// SIMATIC STEP 7 (V5.x) project TF_TACHO_PROJECT
// CPU: CPU 315-2 DP
// station: Hardware
// station: SIMATIC 300
// station: P_ADR_BUS
// station: _S7H_BUSSYSTEM_CT
// program: S7 Program(1)

SYMBOL_TABLE
"DB_Entradas_Proceso"	DB 1	DB 1
"DB_Entradas_HMI"	DB 2	DB 2
"DB_Salidas_Proceso"	DB 3	DB 3
"DB_Salidas_HMI"	DB 4	DB 4
"DB_Flags_Fallas"	DB 5	DB 5
"DB_Aux"	DB 6	DB 6	// DB de variables auxiliares
"DB_Grafo_Marcha"	DB 7	FB 1
"DB_Grafo_ON_OFF"	DB 8	FB 2
"DB_Grafo_PID"	DB 9	FB 3
"DB_CTRL_GRAFOS"	DB 10	DB 10	// DB Global de estados y transiciones de grafos
"DB_PID"	DB 11	FB 41
"FB_Grafo_Marcha"	FB 1	FB 1
"FB_Grafo_ON_OFF"	FB 2	FB 2
"FB_Grafo_PID"	FB 3	FB 3
"CONT_C"	FB 41	FB 41	// Continuous Control
"FC_Init_constantes"	FC 1	FC 1
"FC_Manejo_Entradas_Proc"	FC 2	FC 2
"FC_Manejo_Entradas_HMI"	FC 3	FC 3
"FC_Modos_Operacion"	FC 4	FC 4
"FC_Calculo_Var_Aux"	FC 5	FC 5	// Funcion que calcula variables aux.
"FC_Adm_Fallas"	FC 6	FC 6	// Funcion que verifica fallas del sistema
"FC_Recuperacion_Fallas"	FC 7	FC 7	// Recuperacion automatica de fallas
"FC_Ctrl_ON_OFF"	FC 8	FC 8
"FC_Ctrl_PID"	FC 9	FC 9
"FC_Ctrl_Marcha"	FC 10	FC 10
"FC_Ejecucion_PID"	FC 11	FC 11
"G7_STD_3"	FC 72	FC 72
"SCALE"	FC 105	FC 105	// Scaling Values
"UNSCALE"	FC 106	FC 106	// Unscaling Values
"FALLA_BMB"	I 1.0	BOOL	// Señal (simulada) de falla de bomba
"NIV_SENS"	IW 0	INT	// Nivel sensado del liquido en el tacho (Cuentas)
"FALSE"	M 0.0	BOOL
"TRUE"	M 0.1	BOOL
"ALTURA_TACHO"	MD 1	REAL	// Altura del tacho (cm)
"NIVEL_ALTO"	MD 3	REAL	// Nivel maximo de agua en el tacho
"NIVEL_BAJO"	MD 5	REAL	// Minimo nivel de agua en el tacho
"Programa Principal"	OB 1	OB 1
"CYC_INT5"	OB 35	OB 35	// Cyclic Interrupt 5
"SALIDA_HL"	Q 4.0	BOOL	// Indicacion de nivel alto (HL)
"SALIDA_LL"	Q 4.1	BOOL	// Indicación de nivel bajo (LL)
"LUZ_MODO_OPER"	Q 4.2	BOOL	// Indicacion del modo de operacion (MANUAL-ON/OFF-PID)
"BMB_CARGA"	QW 0	WORD	// Señal de actuación sobre la bomba de carga del sistema. Rango entre 0 y 5 V.
"BMB_PERT"	QW 2	WORD	// Señal de actuación sobre la bomba de perturbación (vaciado) del sistema.
"TIME_TCK"	SFC 64	SFC 64	// Read the System Time
"VAT_SIM"	VAT 1	
END_SYMBOL_TABLE

FUNCTION_BLOCK "FB_Grafo_Marcha"	// FB 1
TITLE = S7GRAPH V4 FB
//Block comment
VERSION : 0.1
VAR_INPUT
  OFF_SQ : BOOL ;
  INIT_SQ : BOOL ;
  ACK_EF : BOOL ;
  S_PREV : BOOL ;
  S_NEXT : BOOL ;
  SW_AUTO : BOOL ;
  SW_TAP : BOOL ;
  SW_MAN : BOOL ;
  S_SEL : INT ;
  S_ON : BOOL ;
  S_OFF : BOOL ;
  T_PUSH : BOOL ;
END_VAR
VAR_OUTPUT
  S_NO : INT ;
  S_MORE : BOOL ;
  S_ACTIVE : BOOL ;
  ERR_FLT : BOOL ;
  AUTO_ON : BOOL ;
  TAP_ON : BOOL ;
  MAN_ON : BOOL ;
END_VAR
VAR
  G7T : ARRAY  [0 .. 3 ] OF STRUCT
   TV : BOOL ;
   TT : BOOL ;
   TS : BOOL ;
   CF_IV : BOOL ;
   TNO : INT ;
   CRIT : DWORD ;
   CRIT_OLD : DWORD ;
   CRIT_FLT : DWORD ;
  END_STRUCT ;
  G7S : ARRAY  [0 .. 3 ] OF STRUCT
   S1 : BOOL ;
   L1 : BOOL ;
   V1 : BOOL ;
   R1 : BOOL ;
   A1 : BOOL ;
   S0 : BOOL ;
   L0 : BOOL ;
   V0 : BOOL ;
   X : BOOL ;
   LA : BOOL ;
   VA : BOOL ;
   RA : BOOL ;
   AA : BOOL ;
   SS : BOOL ;
   LS : BOOL ;
   VS : BOOL ;
   SNO : INT ;
   T : TIME ;
   U : TIME ;
   CRIT_LOC : DWORD ;
   CRIT_LOC_ERR : DWORD ;
   CRIT_SUP : DWORD ;
   SM : BOOL ;
   LP : BOOL ;
   LN : BOOL ;
   VP : BOOL ;
   VN : BOOL ;
   H_IL_ERR : BYTE ;
   H_SV_FLT : BYTE ;
   RESERVED : DWORD ;
  END_STRUCT ;
  TVX : ARRAY  [0 .. 2 ] OF BYTE  := B#16#1;
  TTX : ARRAY  [0 .. 2 ] OF BYTE  := B#16#1;
  TSX : ARRAY  [0 .. 2 ] OF BYTE  := B#16#1;
  S00X : ARRAY  [0 .. 2 ] OF BYTE  := B#16#1;
  SOFFX : ARRAY  [0 .. 2 ] OF BYTE  := B#16#1;
  SONX : ARRAY  [0 .. 2 ] OF BYTE  := B#16#1;
  SAX : ARRAY  [0 .. 2 ] OF BYTE  := B#16#1;
  SERRX : ARRAY  [0 .. 4 ] OF BYTE  := B#16#1;
  SMX : ARRAY  [0 .. 4 ] OF BYTE  := B#16#1;
  S0X : ARRAY  [0 .. 4 ] OF BYTE  := B#16#1;
  S1X : ARRAY  [0 .. 4 ] OF BYTE  := B#16#1;
  S_DISPLAY : INT ;
  S_SEL_OLD : INT ;
  S_DISPIDX : BYTE ;
  T_DISPIDX : BYTE ;
  MOPEDGE : STRUCT
   AUTO : BOOL ;
   MAN : BOOL ;
   TAP : BOOL ;
   TOP : BOOL ;
   RES1 : BOOL ;
   RES2 : BOOL ;
   RES3 : BOOL ;
   RES4 : BOOL ;
   LOCK : BOOL ;
   SUP : BOOL ;
   ACKREQ : BOOL ;
   SSKIP : BOOL ;
   OFF : BOOL ;
   INIT : BOOL ;
   HALT : BOOL ;
   TMS_HALT : BOOL ;
   OPS_ZERO : BOOL ;
   SACT_DISP : BOOL ;
   SEF_DISP : BOOL ;
   SALL_DISP : BOOL ;
   S_PREV : BOOL ;
   S_NEXT : BOOL ;
   S_SELOK : BOOL ;
   S_ON : BOOL ;
   S_OFF : BOOL ;
   T_PUSH : BOOL ;
   REG : BOOL ;
   ACK : BOOL ;
   IL_PERM : BOOL ;
   T_PERM : BOOL ;
   ILP_MAN : BOOL ;
  END_STRUCT ;
  MOP : STRUCT
   AUTO : BOOL  := TRUE;
   MAN : BOOL ;
   TAP : BOOL ;
   TOP : BOOL ;
   RES1 : BOOL ;
   RES2 : BOOL ;
   RES3 : BOOL ;
   RES4 : BOOL ;
   LOCK : BOOL  := TRUE;
   SUP : BOOL  := TRUE;
   ACKREQ : BOOL  := TRUE;
   SSKIP : BOOL ;
   OFF : BOOL ;
   INIT : BOOL  := TRUE;
   HALT : BOOL ;
   TMS_HALT : BOOL ;
   OPS_ZERO : BOOL ;
   SACT_DISP : BOOL  := TRUE;
   SEF_DISP : BOOL ;
   SALL_DISP : BOOL ;
   S_PREV : BOOL ;
   S_NEXT : BOOL ;
   S_SELOK : BOOL ;
   S_ON : BOOL ;
   S_OFF : BOOL ;
   T_PUSH : BOOL ;
   REG : BOOL ;
   ACK : BOOL ;
   IL_PERM : BOOL ;
   T_PERM : BOOL ;
   ILP_MAN : BOOL ;
  END_STRUCT ;
  TICKS : STRUCT
   DELTA : TIME ;
   OLD : TIME ;
   NEW : TIME ;
  END_STRUCT ;
  SQ_FLAGS : STRUCT
   ERR_FLT : BOOL ;
   ERROR : BOOL ;
   FAULT : BOOL ;
   RT_FAIL : BOOL ;
   NO_SNO : BOOL ;
   NF_OFL : BOOL ;
   SA_OFL : BOOL ;
   TV_OFL : BOOL ;
   MSG_OFL : BOOL ;
   NO_SWI : BOOL ;
   CYC_OP : BOOL ;
   AS_MSG : BOOL ;
   AS_SEND : BOOL ;
   SQ_BUSY : BOOL ;
   SA_BUSY : BOOL ;
   AS_SIG : BOOL ;
  END_STRUCT ;
  S_PTR : DWORD  := DW#16#250;
  S_PTR2 : DWORD ;
  S_PTR3 : DWORD  := DW#16#7C0;
  S_PTR4 : DWORD  := DW#16#790;
  T_PTR : DWORD  := DW#16#760;
  C_AR2 : DWORD ;
  M_FBDB : DWORD  := DW#16#10000;
  M_SNO : WORD ;
  M_EVID : WORD ;
  M_EVIL : DWORD ;
  M_EVSV : DWORD ;
  M_EV : DWORD  := DW#16#6D0;
  CRIT : ARRAY  [0 .. 31 ] OF BOOL ;
  S_START : BYTE ;
  S_IDX : BYTE ;
  S_INT : INT  := 72;
  S_TMP : BYTE ;
  T_START : BYTE ;
  T_IDX : BYTE ;
  T_TMP : BYTE ;
  T_TMP2 : BYTE ;
  TV_POT : BYTE  := B#16#6;
  RETURN1 : BYTE ;
  RETURN2 : BYTE ;
  SINI : ARRAY  [0 .. 2 ] OF BYTE  := B#16#2, B#16#1;
  LSTT : ARRAY  [0 .. 3 ] OF BYTE  := B#16#0, B#16#0, B#16#0, B#16#2;
  ATAJ : ARRAY  [0 .. 3 ] OF BYTE  := B#16#0, B#16#1, B#16#2, B#16#3;
  ATAB : ARRAY  [0 .. 3 ] OF BYTE  := B#16#0, B#16#1, B#16#2, B#16#3;
  PSTT : ARRAY  [0 .. 3 ] OF BYTE  := B#16#0, B#16#1, B#16#2, B#16#3;
  NSTT : ARRAY  [0 .. 3 ] OF BYTE  := B#16#1, B#16#2, B#16#3, B#16#2;
  ASSJ : ARRAY  [0 .. 3 ] OF BYTE  := B#16#0, B#16#1, B#16#2, B#16#3;
  ASSB : ARRAY  [0 .. 3 ] OF BYTE  := B#16#0, B#16#1, B#16#2, B#16#3;
  PTTS : ARRAY  [0 .. 3 ] OF BYTE  := B#16#0, B#16#0, B#16#1, B#16#2;
  NTTS : ARRAY  [0 .. 3 ] OF BYTE  := B#16#0, B#16#1, B#16#2, B#16#3;
  PRE_CNT : WORD ;
  POST_CNT : WORD ;
  ADR_COND : WORD ;
  MAX_TVAL : BYTE  := B#16#1;
  MAX_SACT : BYTE  := B#16#1;
  MAX_CRIT : BYTE  := B#16#4;
  T_CNT : BYTE  := B#16#3;
  SUP_CNT : BYTE ;
  LOCK_CNT : BYTE ;
  S_CNT : BYTE  := B#16#3;
  SQ_CNT : BYTE  := B#16#1;
  PRS_INPAR : DWORD  := DW#16#E000F6C8;
  PRS_OUTPAR : DWORD  := DW#16#E000800D;
  GC_FLAGS : STRUCT
   T_MACH : WORD  := W#16#EB;
   COND_ED : WORD  := W#16#E3;
   W_LEVEL : WORD  := W#16#D5;
   AS_MSG : WORD ;
   FB_IF : WORD  := W#16#FC;
   SSB : WORD  := W#16#105;
   CRIT_AVAIL : BOOL ;
   SSKIP_AVAIL : BOOL  := TRUE;
   SSKIP_ON : BOOL ;
   ACK_REQ : BOOL  := TRUE;
   SYNC_AVAIL : BOOL ;
   ILP_MAN : BOOL ;
  END_STRUCT ;
  G7_FBMARK : BYTE  := B#16#25;
  G7_RELEASE : BYTE  := B#16#2A;
  G7_ID2 : BYTE  := B#16#37;
  G7_ID1 : BYTE  := B#16#47;
END_VAR
BEGIN
// body was compiled from an S7-GRAPH chart; compiled code not shown
END_FUNCTION_BLOCK

FUNCTION_BLOCK "FB_Grafo_ON_OFF"	// FB 2
TITLE = S7GRAPH V4 FB
//Block comment
VERSION : 0.1
VAR_INPUT
  OFF_SQ : BOOL ;
  INIT_SQ : BOOL ;
  ACK_EF : BOOL ;
  S_PREV : BOOL ;
  S_NEXT : BOOL ;
  SW_AUTO : BOOL ;
  SW_TAP : BOOL ;
  SW_MAN : BOOL ;
  S_SEL : INT ;
  S_ON : BOOL ;
  S_OFF : BOOL ;
  T_PUSH : BOOL ;
END_VAR
VAR_OUTPUT
  S_NO : INT ;
  S_MORE : BOOL ;
  S_ACTIVE : BOOL ;
  ERR_FLT : BOOL ;
  AUTO_ON : BOOL ;
  TAP_ON : BOOL ;
  MAN_ON : BOOL ;
END_VAR
VAR
  G7T : ARRAY  [0 .. 3 ] OF STRUCT
   TV : BOOL ;
   TT : BOOL ;
   TS : BOOL ;
   CF_IV : BOOL ;
   TNO : INT ;
   CRIT : DWORD ;
   CRIT_OLD : DWORD ;
   CRIT_FLT : DWORD ;
  END_STRUCT ;
  G7S : ARRAY  [0 .. 3 ] OF STRUCT
   S1 : BOOL ;
   L1 : BOOL ;
   V1 : BOOL ;
   R1 : BOOL ;
   A1 : BOOL ;
   S0 : BOOL ;
   L0 : BOOL ;
   V0 : BOOL ;
   X : BOOL ;
   LA : BOOL ;
   VA : BOOL ;
   RA : BOOL ;
   AA : BOOL ;
   SS : BOOL ;
   LS : BOOL ;
   VS : BOOL ;
   SNO : INT ;
   T : TIME ;
   U : TIME ;
   CRIT_LOC : DWORD ;
   CRIT_LOC_ERR : DWORD ;
   CRIT_SUP : DWORD ;
   SM : BOOL ;
   LP : BOOL ;
   LN : BOOL ;
   VP : BOOL ;
   VN : BOOL ;
   H_IL_ERR : BYTE ;
   H_SV_FLT : BYTE ;
   RESERVED : DWORD ;
  END_STRUCT ;
  TVX : ARRAY  [0 .. 2 ] OF BYTE  := B#16#1;
  TTX : ARRAY  [0 .. 2 ] OF BYTE  := B#16#1;
  TSX : ARRAY  [0 .. 2 ] OF BYTE  := B#16#1;
  S00X : ARRAY  [0 .. 2 ] OF BYTE  := B#16#1;
  SOFFX : ARRAY  [0 .. 2 ] OF BYTE  := B#16#1;
  SONX : ARRAY  [0 .. 2 ] OF BYTE  := B#16#1;
  SAX : ARRAY  [0 .. 2 ] OF BYTE  := B#16#1;
  SERRX : ARRAY  [0 .. 4 ] OF BYTE  := B#16#1;
  SMX : ARRAY  [0 .. 4 ] OF BYTE  := B#16#1;
  S0X : ARRAY  [0 .. 4 ] OF BYTE  := B#16#1;
  S1X : ARRAY  [0 .. 4 ] OF BYTE  := B#16#1;
  S_DISPLAY : INT ;
  S_SEL_OLD : INT ;
  S_DISPIDX : BYTE ;
  T_DISPIDX : BYTE ;
  MOPEDGE : STRUCT
   AUTO : BOOL ;
   MAN : BOOL ;
   TAP : BOOL ;
   TOP : BOOL ;
   RES1 : BOOL ;
   RES2 : BOOL ;
   RES3 : BOOL ;
   RES4 : BOOL ;
   LOCK : BOOL ;
   SUP : BOOL ;
   ACKREQ : BOOL ;
   SSKIP : BOOL ;
   OFF : BOOL ;
   INIT : BOOL ;
   HALT : BOOL ;
   TMS_HALT : BOOL ;
   OPS_ZERO : BOOL ;
   SACT_DISP : BOOL ;
   SEF_DISP : BOOL ;
   SALL_DISP : BOOL ;
   S_PREV : BOOL ;
   S_NEXT : BOOL ;
   S_SELOK : BOOL ;
   S_ON : BOOL ;
   S_OFF : BOOL ;
   T_PUSH : BOOL ;
   REG : BOOL ;
   ACK : BOOL ;
   IL_PERM : BOOL ;
   T_PERM : BOOL ;
   ILP_MAN : BOOL ;
  END_STRUCT ;
  MOP : STRUCT
   AUTO : BOOL  := TRUE;
   MAN : BOOL ;
   TAP : BOOL ;
   TOP : BOOL ;
   RES1 : BOOL ;
   RES2 : BOOL ;
   RES3 : BOOL ;
   RES4 : BOOL ;
   LOCK : BOOL  := TRUE;
   SUP : BOOL  := TRUE;
   ACKREQ : BOOL  := TRUE;
   SSKIP : BOOL ;
   OFF : BOOL ;
   INIT : BOOL  := TRUE;
   HALT : BOOL ;
   TMS_HALT : BOOL ;
   OPS_ZERO : BOOL ;
   SACT_DISP : BOOL  := TRUE;
   SEF_DISP : BOOL ;
   SALL_DISP : BOOL ;
   S_PREV : BOOL ;
   S_NEXT : BOOL ;
   S_SELOK : BOOL ;
   S_ON : BOOL ;
   S_OFF : BOOL ;
   T_PUSH : BOOL ;
   REG : BOOL ;
   ACK : BOOL ;
   IL_PERM : BOOL ;
   T_PERM : BOOL ;
   ILP_MAN : BOOL ;
  END_STRUCT ;
  TICKS : STRUCT
   DELTA : TIME ;
   OLD : TIME ;
   NEW : TIME ;
  END_STRUCT ;
  SQ_FLAGS : STRUCT
   ERR_FLT : BOOL ;
   ERROR : BOOL ;
   FAULT : BOOL ;
   RT_FAIL : BOOL ;
   NO_SNO : BOOL ;
   NF_OFL : BOOL ;
   SA_OFL : BOOL ;
   TV_OFL : BOOL ;
   MSG_OFL : BOOL ;
   NO_SWI : BOOL ;
   CYC_OP : BOOL ;
   AS_MSG : BOOL ;
   AS_SEND : BOOL ;
   SQ_BUSY : BOOL ;
   SA_BUSY : BOOL ;
   AS_SIG : BOOL ;
  END_STRUCT ;
  S_PTR : DWORD  := DW#16#250;
  S_PTR2 : DWORD ;
  S_PTR3 : DWORD  := DW#16#7C0;
  S_PTR4 : DWORD  := DW#16#790;
  T_PTR : DWORD  := DW#16#760;
  C_AR2 : DWORD ;
  M_FBDB : DWORD  := DW#16#20000;
  M_SNO : WORD ;
  M_EVID : WORD ;
  M_EVIL : DWORD ;
  M_EVSV : DWORD ;
  M_EV : DWORD  := DW#16#6D0;
  CRIT : ARRAY  [0 .. 31 ] OF BOOL ;
  S_START : BYTE ;
  S_IDX : BYTE ;
  S_INT : INT  := 72;
  S_TMP : BYTE ;
  T_START : BYTE ;
  T_IDX : BYTE ;
  T_TMP : BYTE ;
  T_TMP2 : BYTE ;
  TV_POT : BYTE  := B#16#6;
  RETURN1 : BYTE ;
  RETURN2 : BYTE ;
  SINI : ARRAY  [0 .. 2 ] OF BYTE  := B#16#2, B#16#1;
  LSTT : ARRAY  [0 .. 3 ] OF BYTE  := B#16#0, B#16#0, B#16#0, B#16#2;
  ATAJ : ARRAY  [0 .. 3 ] OF BYTE  := B#16#0, B#16#1, B#16#2, B#16#3;
  ATAB : ARRAY  [0 .. 3 ] OF BYTE  := B#16#0, B#16#1, B#16#2, B#16#3;
  PSTT : ARRAY  [0 .. 3 ] OF BYTE  := B#16#0, B#16#1, B#16#2, B#16#3;
  NSTT : ARRAY  [0 .. 3 ] OF BYTE  := B#16#1, B#16#2, B#16#3, B#16#2;
  ASSJ : ARRAY  [0 .. 3 ] OF BYTE  := B#16#0, B#16#1, B#16#2, B#16#3;
  ASSB : ARRAY  [0 .. 3 ] OF BYTE  := B#16#0, B#16#1, B#16#2, B#16#3;
  PTTS : ARRAY  [0 .. 3 ] OF BYTE  := B#16#0, B#16#0, B#16#1, B#16#2;
  NTTS : ARRAY  [0 .. 3 ] OF BYTE  := B#16#0, B#16#1, B#16#2, B#16#3;
  PRE_CNT : WORD ;
  POST_CNT : WORD ;
  ADR_COND : WORD ;
  MAX_TVAL : BYTE  := B#16#1;
  MAX_SACT : BYTE  := B#16#1;
  MAX_CRIT : BYTE  := B#16#4;
  T_CNT : BYTE  := B#16#3;
  SUP_CNT : BYTE ;
  LOCK_CNT : BYTE ;
  S_CNT : BYTE  := B#16#3;
  SQ_CNT : BYTE  := B#16#1;
  PRS_INPAR : DWORD  := DW#16#E000F6C8;
  PRS_OUTPAR : DWORD  := DW#16#E000800D;
  GC_FLAGS : STRUCT
   T_MACH : WORD  := W#16#EB;
   COND_ED : WORD  := W#16#E3;
   W_LEVEL : WORD  := W#16#D5;
   AS_MSG : WORD ;
   FB_IF : WORD  := W#16#FC;
   SSB : WORD  := W#16#105;
   CRIT_AVAIL : BOOL ;
   SSKIP_AVAIL : BOOL  := TRUE;
   SSKIP_ON : BOOL ;
   ACK_REQ : BOOL  := TRUE;
   SYNC_AVAIL : BOOL ;
   ILP_MAN : BOOL ;
  END_STRUCT ;
  G7_FBMARK : BYTE  := B#16#25;
  G7_RELEASE : BYTE  := B#16#2A;
  G7_ID2 : BYTE  := B#16#37;
  G7_ID1 : BYTE  := B#16#47;
END_VAR
BEGIN
// body was compiled from an S7-GRAPH chart; compiled code not shown
END_FUNCTION_BLOCK

FUNCTION_BLOCK "FB_Grafo_PID"	// FB 3
TITLE = S7GRAPH V4 FB
//Block comment
VERSION : 0.1
VAR_INPUT
  OFF_SQ : BOOL ;
  INIT_SQ : BOOL ;
  ACK_EF : BOOL ;
  S_PREV : BOOL ;
  S_NEXT : BOOL ;
  SW_AUTO : BOOL ;
  SW_TAP : BOOL ;
  SW_MAN : BOOL ;
  S_SEL : INT ;
  S_ON : BOOL ;
  S_OFF : BOOL ;
  T_PUSH : BOOL ;
END_VAR
VAR_OUTPUT
  S_NO : INT ;
  S_MORE : BOOL ;
  S_ACTIVE : BOOL ;
  ERR_FLT : BOOL ;
  AUTO_ON : BOOL ;
  TAP_ON : BOOL ;
  MAN_ON : BOOL ;
END_VAR
VAR
  G7T : ARRAY  [0 .. 2 ] OF STRUCT
   TV : BOOL ;
   TT : BOOL ;
   TS : BOOL ;
   CF_IV : BOOL ;
   TNO : INT ;
   CRIT : DWORD ;
   CRIT_OLD : DWORD ;
   CRIT_FLT : DWORD ;
  END_STRUCT ;
  G7S : ARRAY  [0 .. 2 ] OF STRUCT
   S1 : BOOL ;
   L1 : BOOL ;
   V1 : BOOL ;
   R1 : BOOL ;
   A1 : BOOL ;
   S0 : BOOL ;
   L0 : BOOL ;
   V0 : BOOL ;
   X : BOOL ;
   LA : BOOL ;
   VA : BOOL ;
   RA : BOOL ;
   AA : BOOL ;
   SS : BOOL ;
   LS : BOOL ;
   VS : BOOL ;
   SNO : INT ;
   T : TIME ;
   U : TIME ;
   CRIT_LOC : DWORD ;
   CRIT_LOC_ERR : DWORD ;
   CRIT_SUP : DWORD ;
   SM : BOOL ;
   LP : BOOL ;
   LN : BOOL ;
   VP : BOOL ;
   VN : BOOL ;
   H_IL_ERR : BYTE ;
   H_SV_FLT : BYTE ;
   RESERVED : DWORD ;
  END_STRUCT ;
  TVX : ARRAY  [0 .. 2 ] OF BYTE  := B#16#1;
  TTX : ARRAY  [0 .. 2 ] OF BYTE  := B#16#1;
  TSX : ARRAY  [0 .. 2 ] OF BYTE  := B#16#1;
  S00X : ARRAY  [0 .. 2 ] OF BYTE  := B#16#1;
  SOFFX : ARRAY  [0 .. 2 ] OF BYTE  := B#16#1;
  SONX : ARRAY  [0 .. 2 ] OF BYTE  := B#16#1;
  SAX : ARRAY  [0 .. 2 ] OF BYTE  := B#16#1;
  SERRX : ARRAY  [0 .. 3 ] OF BYTE  := B#16#1;
  SMX : ARRAY  [0 .. 3 ] OF BYTE  := B#16#1;
  S0X : ARRAY  [0 .. 3 ] OF BYTE  := B#16#1;
  S1X : ARRAY  [0 .. 3 ] OF BYTE  := B#16#1;
  S_DISPLAY : INT ;
  S_SEL_OLD : INT ;
  S_DISPIDX : BYTE ;
  T_DISPIDX : BYTE ;
  MOPEDGE : STRUCT
   AUTO : BOOL ;
   MAN : BOOL ;
   TAP : BOOL ;
   TOP : BOOL ;
   RES1 : BOOL ;
   RES2 : BOOL ;
   RES3 : BOOL ;
   RES4 : BOOL ;
   LOCK : BOOL ;
   SUP : BOOL ;
   ACKREQ : BOOL ;
   SSKIP : BOOL ;
   OFF : BOOL ;
   INIT : BOOL ;
   HALT : BOOL ;
   TMS_HALT : BOOL ;
   OPS_ZERO : BOOL ;
   SACT_DISP : BOOL ;
   SEF_DISP : BOOL ;
   SALL_DISP : BOOL ;
   S_PREV : BOOL ;
   S_NEXT : BOOL ;
   S_SELOK : BOOL ;
   S_ON : BOOL ;
   S_OFF : BOOL ;
   T_PUSH : BOOL ;
   REG : BOOL ;
   ACK : BOOL ;
   IL_PERM : BOOL ;
   T_PERM : BOOL ;
   ILP_MAN : BOOL ;
  END_STRUCT ;
  MOP : STRUCT
   AUTO : BOOL  := TRUE;
   MAN : BOOL ;
   TAP : BOOL ;
   TOP : BOOL ;
   RES1 : BOOL ;
   RES2 : BOOL ;
   RES3 : BOOL ;
   RES4 : BOOL ;
   LOCK : BOOL  := TRUE;
   SUP : BOOL  := TRUE;
   ACKREQ : BOOL  := TRUE;
   SSKIP : BOOL ;
   OFF : BOOL ;
   INIT : BOOL  := TRUE;
   HALT : BOOL ;
   TMS_HALT : BOOL ;
   OPS_ZERO : BOOL ;
   SACT_DISP : BOOL  := TRUE;
   SEF_DISP : BOOL ;
   SALL_DISP : BOOL ;
   S_PREV : BOOL ;
   S_NEXT : BOOL ;
   S_SELOK : BOOL ;
   S_ON : BOOL ;
   S_OFF : BOOL ;
   T_PUSH : BOOL ;
   REG : BOOL ;
   ACK : BOOL ;
   IL_PERM : BOOL ;
   T_PERM : BOOL ;
   ILP_MAN : BOOL ;
  END_STRUCT ;
  TICKS : STRUCT
   DELTA : TIME ;
   OLD : TIME ;
   NEW : TIME ;
  END_STRUCT ;
  SQ_FLAGS : STRUCT
   ERR_FLT : BOOL ;
   ERROR : BOOL ;
   FAULT : BOOL ;
   RT_FAIL : BOOL ;
   NO_SNO : BOOL ;
   NF_OFL : BOOL ;
   SA_OFL : BOOL ;
   TV_OFL : BOOL ;
   MSG_OFL : BOOL ;
   NO_SWI : BOOL ;
   CYC_OP : BOOL ;
   AS_MSG : BOOL ;
   AS_SEND : BOOL ;
   SQ_BUSY : BOOL ;
   SA_BUSY : BOOL ;
   AS_SIG : BOOL ;
  END_STRUCT ;
  S_PTR : DWORD  := DW#16#1D0;
  S_PTR2 : DWORD ;
  S_PTR3 : DWORD  := DW#16#610;
  S_PTR4 : DWORD  := DW#16#5F0;
  T_PTR : DWORD  := DW#16#5D0;
  C_AR2 : DWORD ;
  M_FBDB : DWORD  := DW#16#30000;
  M_SNO : WORD ;
  M_EVID : WORD ;
  M_EVIL : DWORD ;
  M_EVSV : DWORD ;
  M_EV : DWORD  := DW#16#550;
  CRIT : ARRAY  [0 .. 31 ] OF BOOL ;
  S_START : BYTE ;
  S_IDX : BYTE ;
  S_INT : INT  := 72;
  S_TMP : BYTE ;
  T_START : BYTE ;
  T_IDX : BYTE ;
  T_TMP : BYTE ;
  T_TMP2 : BYTE ;
  TV_POT : BYTE  := B#16#6;
  RETURN1 : BYTE ;
  RETURN2 : BYTE ;
  SINI : ARRAY  [0 .. 2 ] OF BYTE  := B#16#2, B#16#1;
  LSTT : ARRAY  [0 .. 2 ] OF BYTE  := B#16#0, B#16#0, B#16#1;
  ATAJ : ARRAY  [0 .. 2 ] OF BYTE  := B#16#0, B#16#1, B#16#2;
  ATAB : ARRAY  [0 .. 2 ] OF BYTE  := B#16#0, B#16#1, B#16#2;
  PSTT : ARRAY  [0 .. 2 ] OF BYTE  := B#16#0, B#16#1, B#16#2;
  NSTT : ARRAY  [0 .. 2 ] OF BYTE  := B#16#1, B#16#2, B#16#1;
  ASSJ : ARRAY  [0 .. 2 ] OF BYTE  := B#16#0, B#16#1, B#16#2;
  ASSB : ARRAY  [0 .. 2 ] OF BYTE  := B#16#0, B#16#1, B#16#2;
  PTTS : ARRAY  [0 .. 2 ] OF BYTE  := B#16#0, B#16#0, B#16#1;
  NTTS : ARRAY  [0 .. 2 ] OF BYTE  := B#16#0, B#16#1, B#16#2;
  PRE_CNT : WORD ;
  POST_CNT : WORD ;
  ADR_COND : WORD ;
  MAX_TVAL : BYTE  := B#16#1;
  MAX_SACT : BYTE  := B#16#1;
  MAX_CRIT : BYTE  := B#16#4;
  T_CNT : BYTE  := B#16#2;
  SUP_CNT : BYTE ;
  LOCK_CNT : BYTE ;
  S_CNT : BYTE  := B#16#2;
  SQ_CNT : BYTE  := B#16#1;
  PRS_INPAR : DWORD  := DW#16#E000F6C8;
  PRS_OUTPAR : DWORD  := DW#16#E000800D;
  GC_FLAGS : STRUCT
   T_MACH : WORD  := W#16#EB;
   COND_ED : WORD  := W#16#E3;
   W_LEVEL : WORD  := W#16#D5;
   AS_MSG : WORD ;
   FB_IF : WORD  := W#16#FC;
   SSB : WORD  := W#16#105;
   CRIT_AVAIL : BOOL ;
   SSKIP_AVAIL : BOOL  := TRUE;
   SSKIP_ON : BOOL ;
   ACK_REQ : BOOL  := TRUE;
   SYNC_AVAIL : BOOL ;
   ILP_MAN : BOOL ;
  END_STRUCT ;
  G7_FBMARK : BYTE  := B#16#25;
  G7_RELEASE : BYTE  := B#16#2A;
  G7_ID2 : BYTE  := B#16#37;
  G7_ID1 : BYTE  := B#16#47;
END_VAR
BEGIN
// body was compiled from an S7-GRAPH chart; compiled code not shown
END_FUNCTION_BLOCK

// FB 41: know-how protected block, not included

FUNCTION "FC_Init_constantes" : VOID	// FC 1
TITLE = Inicializacion de constantes
VERSION : 0.1
BEGIN
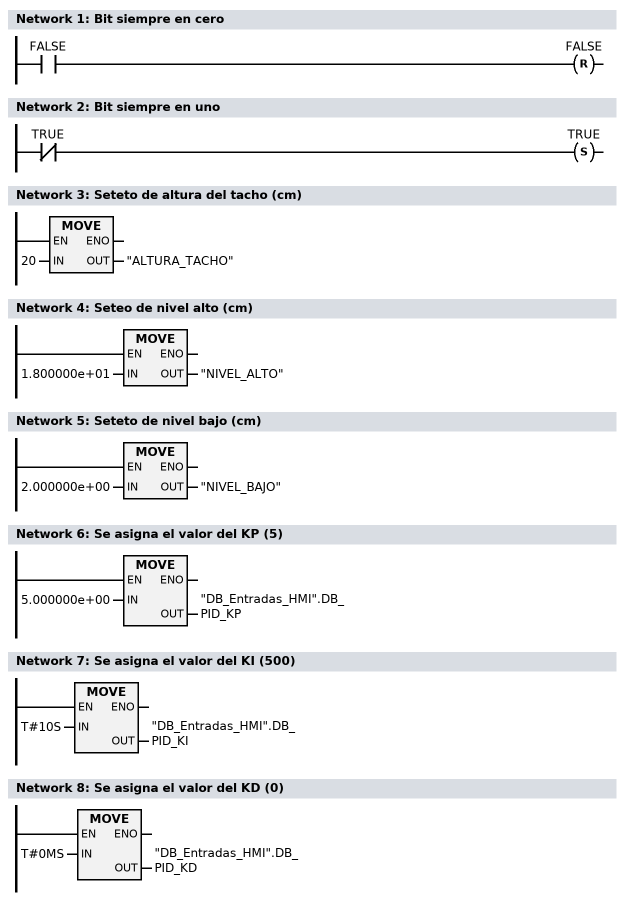
NETWORK
TITLE = Bit siempre en cero
      A     "FALSE";
      R     "FALSE";
NETWORK
TITLE = Bit siempre en uno
      AN    "TRUE";
      S     "TRUE";
NETWORK
TITLE = Seteto de altura del tacho (cm)
      L     20;
      T     "ALTURA_TACHO";
      NOP   0;
NETWORK
TITLE = Seteo de nivel alto (cm)
      L     1.800000e+01;
      T     "NIVEL_ALTO";
      NOP   0;
NETWORK
TITLE = Seteto de nivel bajo (cm)
      L     2.000000e+00;
      T     "NIVEL_BAJO";
      NOP   0;
NETWORK
TITLE = Se asigna el valor del KP (5)
      L     5.000000e+00;
      T     "DB_Entradas_HMI".DB_PID_KP;
      NOP   0;
NETWORK
TITLE = Se asigna el valor del KI (500)
      L     T#10S;
      T     "DB_Entradas_HMI".DB_PID_KI;
      NOP   0;
NETWORK
TITLE = Se asigna el valor del KD (0)
      L     T#0MS;
      T     "DB_Entradas_HMI".DB_PID_KD;
      NOP   0;
END_FUNCTION

FUNCTION "FC_Manejo_Entradas_Proc" : VOID	// FC 2
TITLE = Procesamiento de entradas
VERSION : 0.1
VAR_TEMP
  TMP_NIVEL : INT ;
  TMP_RV : WORD ;
  ES_MAYOR : BOOL ;
  TMP_ENO : BOOL ;
END_VAR
BEGIN
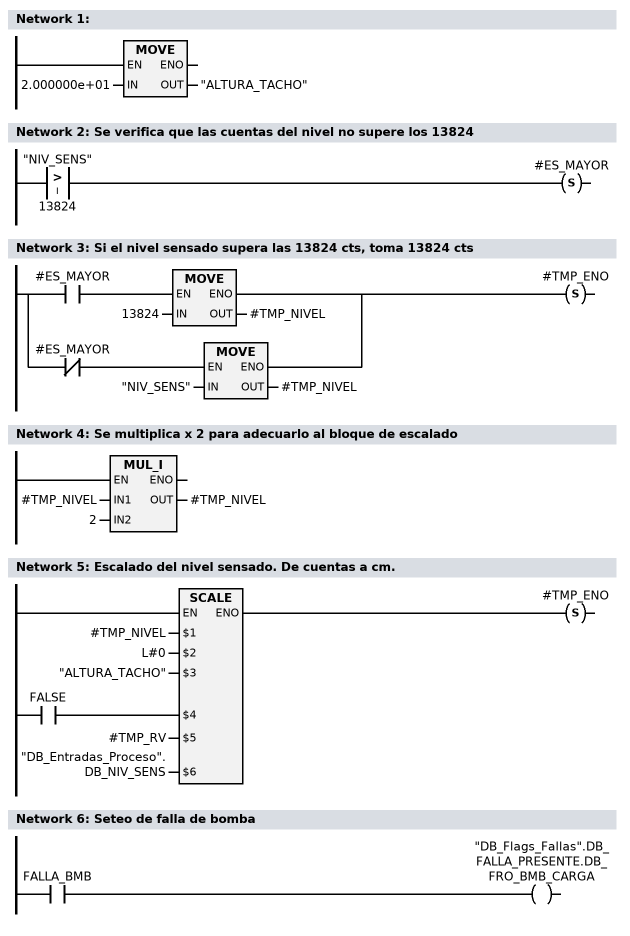
NETWORK
TITLE =
      L     2.000000e+01;
      T     "ALTURA_TACHO";
      NOP   0;
NETWORK
TITLE = Se verifica que las cuentas del nivel no supere los 13824
      L     "NIV_SENS";
      L     13824;
      >I;
      S     #ES_MAYOR;
NETWORK
TITLE = Si el nivel sensado supera las 13824 cts, toma 13824 cts
      O(;
      A     #ES_MAYOR;
      JNB   _001;
      L     13824;
      T     #TMP_NIVEL;
      SET;
      SAVE;
      CLR;
_001: A     BR;
      );
      O(;
      AN    #ES_MAYOR;
      JNB   _002;
      L     "NIV_SENS";
      T     #TMP_NIVEL;
      SET;
      SAVE;
      CLR;
_002: A     BR;
      );
      S     #TMP_ENO;
NETWORK
TITLE = Se multiplica x 2 para adecuarlo al bloque de escalado
      L     #TMP_NIVEL;
      L     2;
      *I;
      T     #TMP_NIVEL;
      NOP   0;
NETWORK
TITLE = Escalado del nivel sensado. De cuentas a cm.
      A     "FALSE";
      =     L 5.0;
      BLD   103;
      CALL  "SCALE" (
           $1                       := #TMP_NIVEL,
           $2                       := L#0,
           $3                       := "ALTURA_TACHO",
           $4                       := L 5.0,
           $5                       := #TMP_RV,
           $6                       := "DB_Entradas_Proceso".DB_NIV_SENS);
      A     BR;
      S     #TMP_ENO;
NETWORK
TITLE = Seteo de falla de bomba
      A     "FALLA_BMB";
      =     "DB_Flags_Fallas".DB_FALLA_PRESENTE.DB_FRO_BMB_CARGA;
END_FUNCTION

FUNCTION "FC_Manejo_Entradas_HMI" : VOID	// FC 3
//Funcion de validacion de las entradas del HMI
VERSION : 0.1
VAR_TEMP
  TMP_MAX_HIST : REAL ;
END_VAR
BEGIN
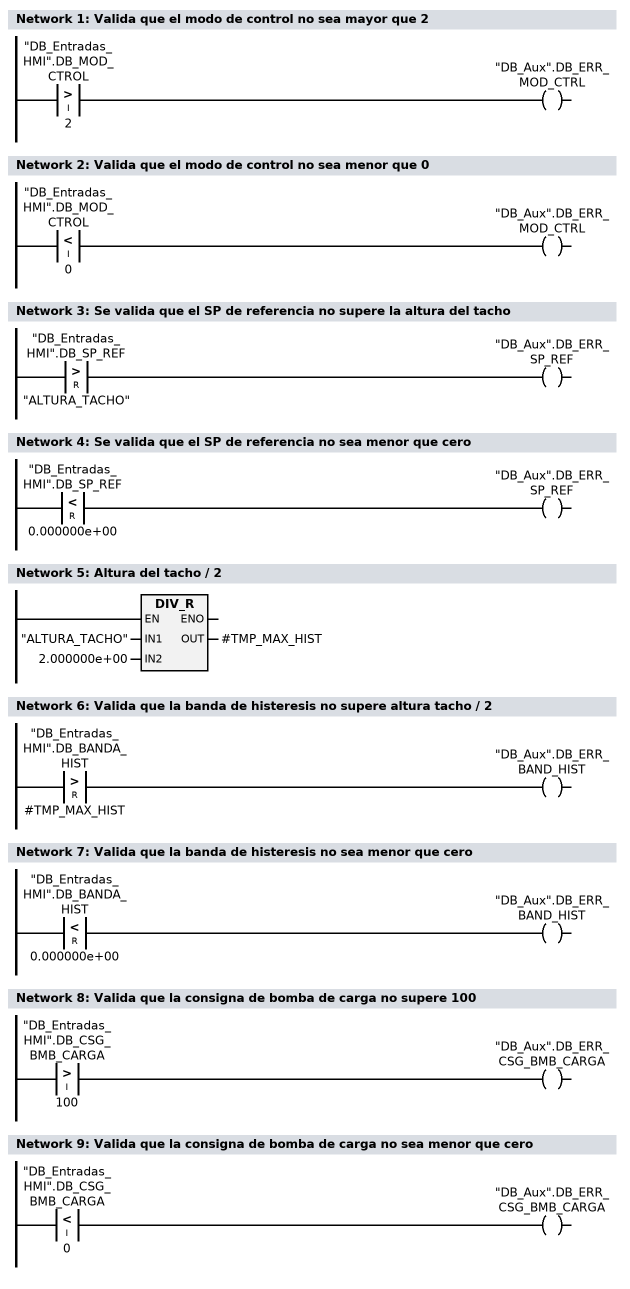
NETWORK
TITLE = Valida que el modo de control no sea mayor que 2
      L     "DB_Entradas_HMI".DB_MOD_CTROL;
      L     2;
      >I;
      =     "DB_Aux".DB_ERR_MOD_CTRL;
NETWORK
TITLE = Valida que el modo de control no sea menor que 0
      L     "DB_Entradas_HMI".DB_MOD_CTROL;
      L     0;
      <I;
      =     "DB_Aux".DB_ERR_MOD_CTRL;
NETWORK
TITLE = Se valida que el SP de referencia no supere la altura del tacho
      L     "DB_Entradas_HMI".DB_SP_REF;
      L     "ALTURA_TACHO";
      >R;
      =     "DB_Aux".DB_ERR_SP_REF;
NETWORK
TITLE = Se valida que el SP de referencia no sea menor que cero
      L     "DB_Entradas_HMI".DB_SP_REF;
      L     0.000000e+00;
      <R;
      =     "DB_Aux".DB_ERR_SP_REF;
NETWORK
TITLE = Altura del tacho / 2
      L     "ALTURA_TACHO";
      L     2.000000e+00;
      /R;
      T     #TMP_MAX_HIST;
      NOP   0;
NETWORK
TITLE = Valida que la banda de histeresis no supere altura tacho / 2
      L     "DB_Entradas_HMI".DB_BANDA_HIST;
      L     #TMP_MAX_HIST;
      >R;
      =     "DB_Aux".DB_ERR_BAND_HIST;
NETWORK
TITLE = Valida que la banda de histeresis no sea menor que cero
      L     "DB_Entradas_HMI".DB_BANDA_HIST;
      L     0.000000e+00;
      <R;
      =     "DB_Aux".DB_ERR_BAND_HIST;
NETWORK
TITLE = Valida que la consigna de bomba de carga no supere 100
      L     "DB_Entradas_HMI".DB_CSG_BMB_CARGA;
      L     100;
      >I;
      =     "DB_Aux".DB_ERR_CSG_BMB_CARGA;
NETWORK
TITLE = Valida que la consigna de bomba de carga no sea menor que cero
      L     "DB_Entradas_HMI".DB_CSG_BMB_CARGA;
      L     0;
      <I;
      =     "DB_Aux".DB_ERR_CSG_BMB_CARGA;
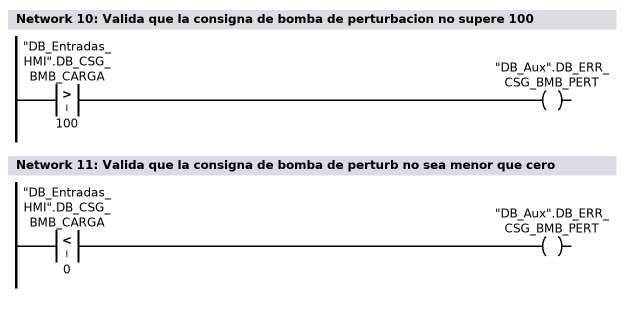
NETWORK
TITLE = Valida que la consigna de bomba de perturbacion no supere 100
      L     "DB_Entradas_HMI".DB_CSG_BMB_CARGA;
      L     100;
      >I;
      =     "DB_Aux".DB_ERR_CSG_BMB_PERT;
NETWORK
TITLE = Valida que la consigna de bomba de perturb no sea menor que cero
      L     "DB_Entradas_HMI".DB_CSG_BMB_CARGA;
      L     0;
      <I;
      =     "DB_Aux".DB_ERR_CSG_BMB_PERT;
END_FUNCTION

FUNCTION "FC_Modos_Operacion" : VOID	// FC 4
VERSION : 0.1
VAR_TEMP
  TMP_SR_MANUAL : BOOL ;	//Temporal usada en el flip flop de manual
  TMP_SR_ONOFF : BOOL ;	//Temporal usada en el flip flop de ON/OFF
  TMP_SR_PID : BOOL ;	//Temporal usada en el flip flop de PID
END_VAR
BEGIN
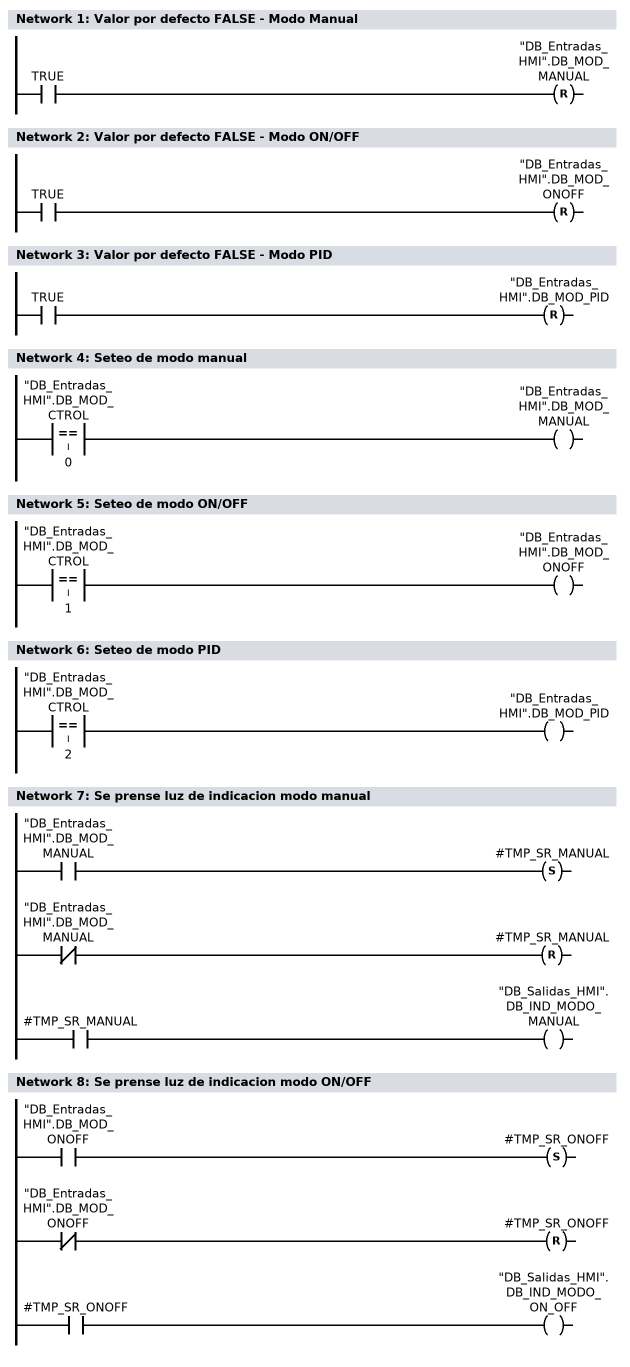
NETWORK
TITLE = Valor por defecto FALSE - Modo Manual
      A     "TRUE";
      R     "DB_Entradas_HMI".DB_MOD_MANUAL;
NETWORK
TITLE = Valor por defecto FALSE - Modo ON/OFF
      A     "TRUE";
      R     "DB_Entradas_HMI".DB_MOD_ONOFF;
NETWORK
TITLE = Valor por defecto FALSE - Modo PID
      A     "TRUE";
      R     "DB_Entradas_HMI".DB_MOD_PID;
NETWORK
TITLE = Seteo de modo manual
      L     "DB_Entradas_HMI".DB_MOD_CTROL;
      L     0;
      ==I;
      =     "DB_Entradas_HMI".DB_MOD_MANUAL;
NETWORK
TITLE = Seteo de modo ON/OFF
      L     "DB_Entradas_HMI".DB_MOD_CTROL;
      L     1;
      ==I;
      =     "DB_Entradas_HMI".DB_MOD_ONOFF;
NETWORK
TITLE = Seteo de modo PID
      L     "DB_Entradas_HMI".DB_MOD_CTROL;
      L     2;
      ==I;
      =     "DB_Entradas_HMI".DB_MOD_PID;
NETWORK
TITLE = Se prense luz de indicacion modo manual
      A     "DB_Entradas_HMI".DB_MOD_MANUAL;
      S     #TMP_SR_MANUAL;
      AN    "DB_Entradas_HMI".DB_MOD_MANUAL;
      R     #TMP_SR_MANUAL;
      A     #TMP_SR_MANUAL;
      =     "DB_Salidas_HMI".DB_IND_MODO_MANUAL;
NETWORK
TITLE = Se prense luz de indicacion modo ON/OFF
      A     "DB_Entradas_HMI".DB_MOD_ONOFF;
      S     #TMP_SR_ONOFF;
      AN    "DB_Entradas_HMI".DB_MOD_ONOFF;
      R     #TMP_SR_ONOFF;
      A     #TMP_SR_ONOFF;
      =     "DB_Salidas_HMI".DB_IND_MODO_ON_OFF;
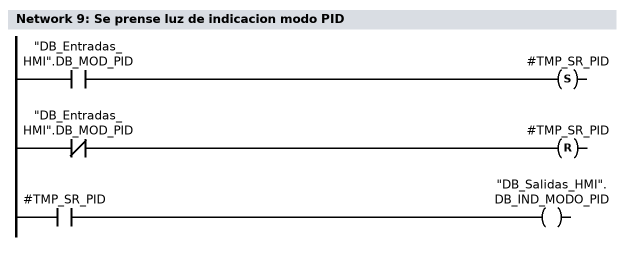
NETWORK
TITLE = Se prense luz de indicacion modo PID
      A     "DB_Entradas_HMI".DB_MOD_PID;
      S     #TMP_SR_PID;
      AN    "DB_Entradas_HMI".DB_MOD_PID;
      R     #TMP_SR_PID;
      A     #TMP_SR_PID;
      =     "DB_Salidas_HMI".DB_IND_MODO_PID;
END_FUNCTION

FUNCTION "FC_Calculo_Var_Aux" : VOID	// FC 5
VERSION : 0.1
VAR_TEMP
  TMP_AUX_DI : DINT ;
  TMP_AUX_R : REAL ;
  TMP_RV : WORD ;
  TMP_RESULT_BAND_HIST : REAL ;
  TMP_FLAG_AUX : BOOL ;
  TMP_SR : BOOL ;
END_VAR
BEGIN
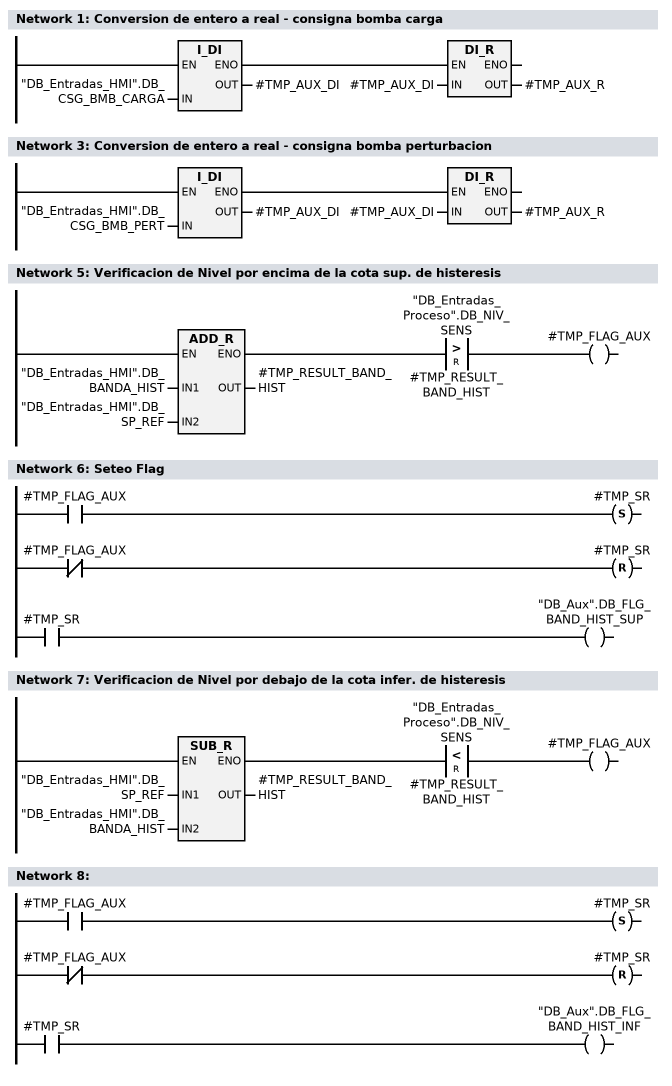
NETWORK
TITLE = Conversion de entero a real - consigna bomba carga
      A(;
      L     "DB_Entradas_HMI".DB_CSG_BMB_CARGA;
      ITD;
      T     #TMP_AUX_DI;
      SET;
      SAVE;
      CLR;
      A     BR;
      );
      JNB   _001;
      L     #TMP_AUX_DI;
      DTR;
      T     #TMP_AUX_R;
_001: NOP   0;
NETWORK
TITLE = Conversion de consigna a cuentas para bomba de cargas
      A(;
      A     "FALSE";
      =     L 15.0;
      BLD   103;
      CALL  "UNSCALE" (
           $1                       := #TMP_AUX_R,
           $2                       := L#1120403456,
           $3                       := L#0,
           $4                       := L 15.0,
           $5                       := #TMP_RV,
           $6                       := "DB_Aux".DB_CTAS_BMB_CARGA);
      A     BR;
      );
      JNB   _002;
      L     "DB_Aux".DB_CTAS_BMB_CARGA;
      L     2;
      /I;
      T     "DB_Aux".DB_CTAS_BMB_CARGA;
_002: NOP   0;
NETWORK
TITLE = Conversion de entero a real - consigna bomba perturbacion
      A(;
      L     "DB_Entradas_HMI".DB_CSG_BMB_PERT;
      ITD;
      T     #TMP_AUX_DI;
      SET;
      SAVE;
      CLR;
      A     BR;
      );
      JNB   _003;
      L     #TMP_AUX_DI;
      DTR;
      T     #TMP_AUX_R;
_003: NOP   0;
NETWORK
TITLE = Conversion de consigna a cuentas para bomba de perturbacion
      A(;
      A     "FALSE";
      =     L 15.0;
      BLD   103;
      CALL  "UNSCALE" (
           $1                       := #TMP_AUX_R,
           $2                       := L#1120403456,
           $3                       := L#0,
           $4                       := L 15.0,
           $5                       := #TMP_RV,
           $6                       := "DB_Aux".DB_CTAS_BMB_PERT);
      A     BR;
      );
      JNB   _004;
      L     "DB_Aux".DB_CTAS_BMB_PERT;
      L     2;
      /I;
      T     "DB_Aux".DB_CTAS_BMB_PERT;
_004: NOP   0;
NETWORK
TITLE = Verificacion de Nivel por encima de la cota sup. de histeresis
      A(;
      L     "DB_Entradas_HMI".DB_BANDA_HIST;
      L     "DB_Entradas_HMI".DB_SP_REF;
      +R;
      T     #TMP_RESULT_BAND_HIST;
      AN    OV;
      SAVE;
      CLR;
      A     BR;
      );
      A(;
      L     "DB_Entradas_Proceso".DB_NIV_SENS;
      L     #TMP_RESULT_BAND_HIST;
      >R;
      );
      =     #TMP_FLAG_AUX;
NETWORK
TITLE = Seteo Flag
      A     #TMP_FLAG_AUX;
      S     #TMP_SR;
      AN    #TMP_FLAG_AUX;
      R     #TMP_SR;
      A     #TMP_SR;
      =     "DB_Aux".DB_FLG_BAND_HIST_SUP;
NETWORK
TITLE = Verificacion de Nivel por debajo de la cota infer. de histeresis
      A(;
      L     "DB_Entradas_HMI".DB_SP_REF;
      L     "DB_Entradas_HMI".DB_BANDA_HIST;
      -R;
      T     #TMP_RESULT_BAND_HIST;
      AN    OV;
      SAVE;
      CLR;
      A     BR;
      );
      A(;
      L     "DB_Entradas_Proceso".DB_NIV_SENS;
      L     #TMP_RESULT_BAND_HIST;
      <R;
      );
      =     #TMP_FLAG_AUX;
NETWORK
TITLE =
      A     #TMP_FLAG_AUX;
      S     #TMP_SR;
      AN    #TMP_FLAG_AUX;
      R     #TMP_SR;
      A     #TMP_SR;
      =     "DB_Aux".DB_FLG_BAND_HIST_INF;
END_FUNCTION

FUNCTION "FC_Adm_Fallas" : VOID	// FC 6
VERSION : 0.1
VAR_TEMP
  FLG_MAYOR_MAX : BOOL ;
  FLG_MENOR_MIN : BOOL ;
  TMP_SR : BOOL ;
END_VAR
BEGIN
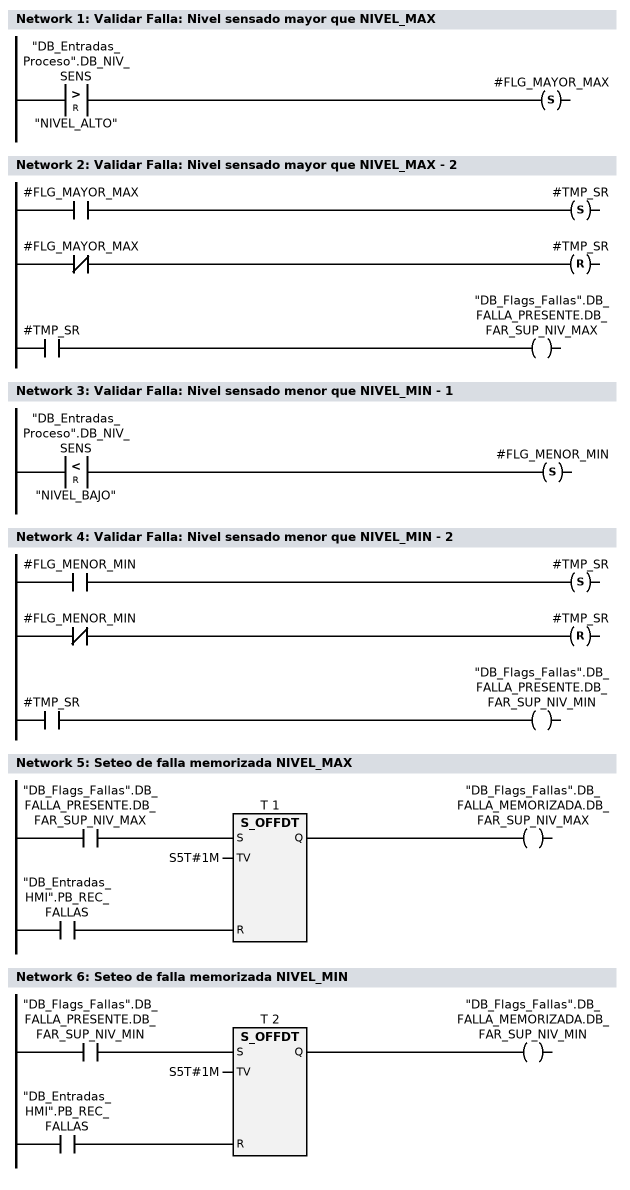
NETWORK
TITLE = Validar Falla: Nivel sensado mayor que NIVEL_MAX
      L     "DB_Entradas_Proceso".DB_NIV_SENS;
      L     "NIVEL_ALTO";
      >R;
      S     #FLG_MAYOR_MAX;
NETWORK
TITLE = Validar Falla: Nivel sensado mayor que NIVEL_MAX - 2
      A     #FLG_MAYOR_MAX;
      S     #TMP_SR;
      AN    #FLG_MAYOR_MAX;
      R     #TMP_SR;
      A     #TMP_SR;
      =     "DB_Flags_Fallas".DB_FALLA_PRESENTE.DB_FAR_SUP_NIV_MAX;
NETWORK
TITLE = Validar Falla: Nivel sensado menor que NIVEL_MIN - 1
      L     "DB_Entradas_Proceso".DB_NIV_SENS;
      L     "NIVEL_BAJO";
      <R;
      S     #FLG_MENOR_MIN;
NETWORK
TITLE = Validar Falla: Nivel sensado menor que NIVEL_MIN - 2
      A     #FLG_MENOR_MIN;
      S     #TMP_SR;
      AN    #FLG_MENOR_MIN;
      R     #TMP_SR;
      A     #TMP_SR;
      =     "DB_Flags_Fallas".DB_FALLA_PRESENTE.DB_FAR_SUP_NIV_MIN;
NETWORK
TITLE = Seteo de falla memorizada NIVEL_MAX
      A     "DB_Flags_Fallas".DB_FALLA_PRESENTE.DB_FAR_SUP_NIV_MAX;
      L     S5T#1M;
      SF    T 1;
      A     "DB_Entradas_HMI".PB_REC_FALLAS;
      R     T 1;
      NOP   0;
      NOP   0;
      A     T 1;
      =     "DB_Flags_Fallas".DB_FALLA_MEMORIZADA.DB_FAR_SUP_NIV_MAX;
NETWORK
TITLE = Seteo de falla memorizada NIVEL_MIN
      A     "DB_Flags_Fallas".DB_FALLA_PRESENTE.DB_FAR_SUP_NIV_MIN;
      L     S5T#1M;
      SF    T 2;
      A     "DB_Entradas_HMI".PB_REC_FALLAS;
      R     T 2;
      NOP   0;
      NOP   0;
      A     T 2;
      =     "DB_Flags_Fallas".DB_FALLA_MEMORIZADA.DB_FAR_SUP_NIV_MIN;
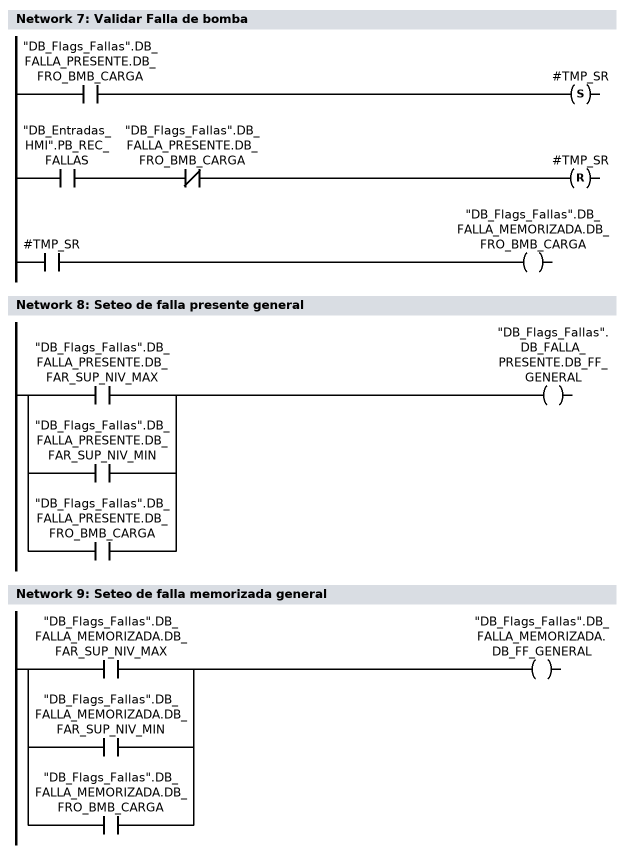
NETWORK
TITLE = Validar Falla de bomba
      A     "DB_Flags_Fallas".DB_FALLA_PRESENTE.DB_FRO_BMB_CARGA;
      S     #TMP_SR;
      A     "DB_Entradas_HMI".PB_REC_FALLAS;
      AN    "DB_Flags_Fallas".DB_FALLA_PRESENTE.DB_FRO_BMB_CARGA;
      R     #TMP_SR;
      A     #TMP_SR;
      =     "DB_Flags_Fallas".DB_FALLA_MEMORIZADA.DB_FRO_BMB_CARGA;
NETWORK
TITLE = Seteo de falla presente general
      O     "DB_Flags_Fallas".DB_FALLA_PRESENTE.DB_FAR_SUP_NIV_MAX;
      O     "DB_Flags_Fallas".DB_FALLA_PRESENTE.DB_FAR_SUP_NIV_MIN;
      O     "DB_Flags_Fallas".DB_FALLA_PRESENTE.DB_FRO_BMB_CARGA;
      =     "DB_Flags_Fallas".DB_FALLA_PRESENTE.DB_FF_GENERAL;
NETWORK
TITLE = Seteo de falla memorizada general
      O     "DB_Flags_Fallas".DB_FALLA_MEMORIZADA.DB_FAR_SUP_NIV_MAX;
      O     "DB_Flags_Fallas".DB_FALLA_MEMORIZADA.DB_FAR_SUP_NIV_MIN;
      O     "DB_Flags_Fallas".DB_FALLA_MEMORIZADA.DB_FRO_BMB_CARGA;
      =     "DB_Flags_Fallas".DB_FALLA_MEMORIZADA.DB_FF_GENERAL;
END_FUNCTION

FUNCTION "FC_Recuperacion_Fallas" : VOID	// FC 7
VERSION : 0.1
BEGIN
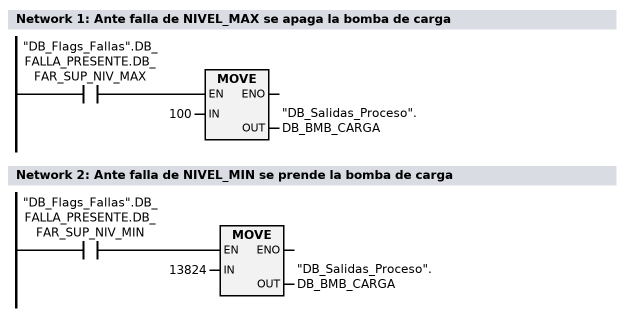
NETWORK
TITLE = Ante falla de NIVEL_MAX se apaga la bomba de carga
      A     "DB_Flags_Fallas".DB_FALLA_PRESENTE.DB_FAR_SUP_NIV_MAX;
      JNB   _001;
      L     100;
      T     "DB_Salidas_Proceso".DB_BMB_CARGA;
_001: NOP   0;
NETWORK
TITLE = Ante falla de NIVEL_MIN se prende la bomba de carga
      A     "DB_Flags_Fallas".DB_FALLA_PRESENTE.DB_FAR_SUP_NIV_MIN;
      JNB   _002;
      L     13824;
      T     "DB_Salidas_Proceso".DB_BMB_CARGA;
_002: NOP   0;
END_FUNCTION

FUNCTION "FC_Ctrl_ON_OFF" : VOID	// FC 8
VERSION : 0.1
BEGIN
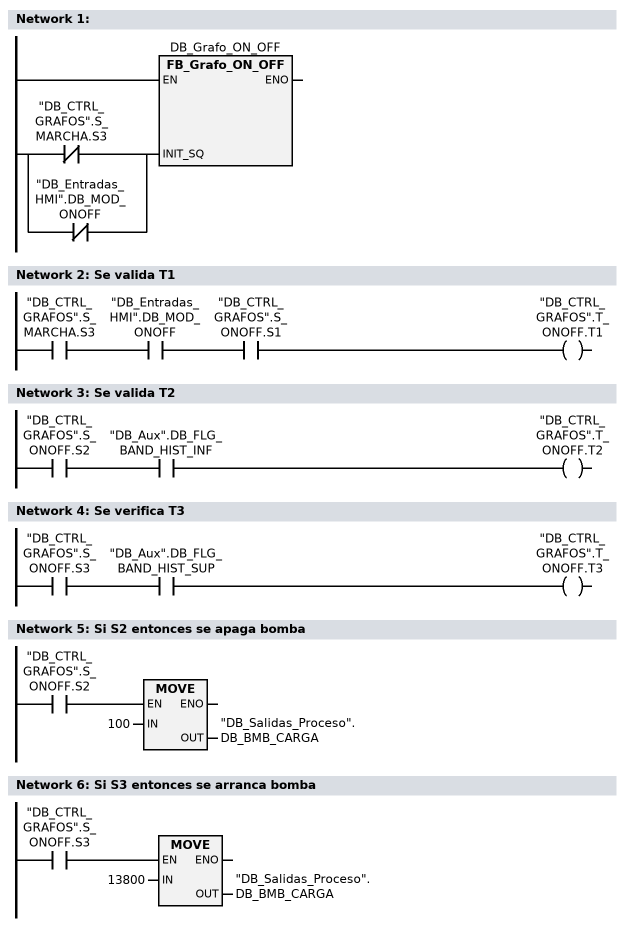
NETWORK
TITLE =
      A(;
      ON    "DB_CTRL_GRAFOS".S_MARCHA.S3;
      ON    "DB_Entradas_HMI".DB_MOD_ONOFF;
      );
      =     L 0.1;
      BLD   103;
      CALL  "FB_Grafo_ON_OFF" , "DB_Grafo_ON_OFF" (
           INIT_SQ                  := L 0.1);
      NOP   0;
NETWORK
TITLE = Se valida T1
      A     "DB_CTRL_GRAFOS".S_MARCHA.S3;
      A     "DB_Entradas_HMI".DB_MOD_ONOFF;
      A     "DB_CTRL_GRAFOS".S_ONOFF.S1;
      =     "DB_CTRL_GRAFOS".T_ONOFF.T1;
NETWORK
TITLE = Se valida T2
      A     "DB_CTRL_GRAFOS".S_ONOFF.S2;
      A     "DB_Aux".DB_FLG_BAND_HIST_INF;
      =     "DB_CTRL_GRAFOS".T_ONOFF.T2;
NETWORK
TITLE = Se verifica T3
      A     "DB_CTRL_GRAFOS".S_ONOFF.S3;
      A     "DB_Aux".DB_FLG_BAND_HIST_SUP;
      =     "DB_CTRL_GRAFOS".T_ONOFF.T3;
NETWORK
TITLE = Si S2 entonces se apaga bomba
      A     "DB_CTRL_GRAFOS".S_ONOFF.S2;
      JNB   _001;
      L     100;
      T     "DB_Salidas_Proceso".DB_BMB_CARGA;
_001: NOP   0;
NETWORK
TITLE = Si S3 entonces se arranca bomba
      A     "DB_CTRL_GRAFOS".S_ONOFF.S3;
      JNB   _002;
      L     13800;
      T     "DB_Salidas_Proceso".DB_BMB_CARGA;
_002: NOP   0;
END_FUNCTION

FUNCTION "FC_Ctrl_PID" : VOID	// FC 9
VERSION : 0.1
BEGIN
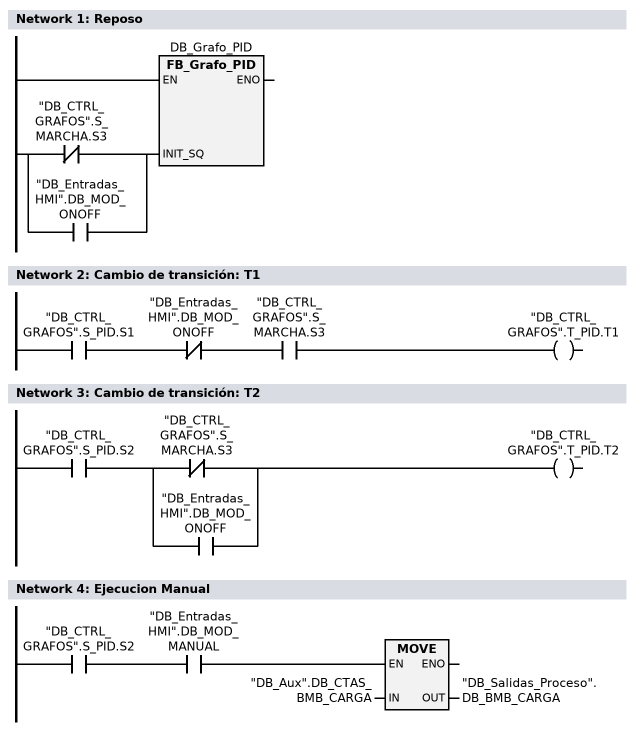
NETWORK
TITLE = Reposo
      A(;
      ON    "DB_CTRL_GRAFOS".S_MARCHA.S3;
      O     "DB_Entradas_HMI".DB_MOD_ONOFF;
      );
      =     L 0.1;
      BLD   103;
      CALL  "FB_Grafo_PID" , "DB_Grafo_PID" (
           INIT_SQ                  := L 0.1);
      NOP   0;
NETWORK
TITLE = Cambio de transición: T1
      A     "DB_CTRL_GRAFOS".S_PID.S1;
      AN    "DB_Entradas_HMI".DB_MOD_ONOFF;
      A     "DB_CTRL_GRAFOS".S_MARCHA.S3;
      =     "DB_CTRL_GRAFOS".T_PID.T1;
NETWORK
TITLE = Cambio de transición: T2
      A     "DB_CTRL_GRAFOS".S_PID.S2;
      A(;
      ON    "DB_CTRL_GRAFOS".S_MARCHA.S3;
      O     "DB_Entradas_HMI".DB_MOD_ONOFF;
      );
      =     "DB_CTRL_GRAFOS".T_PID.T2;
NETWORK
TITLE = Ejecucion Manual
      A     "DB_CTRL_GRAFOS".S_PID.S2;
      A     "DB_Entradas_HMI".DB_MOD_MANUAL;
      JNB   _001;
      L     "DB_Aux".DB_CTAS_BMB_CARGA;
      T     "DB_Salidas_Proceso".DB_BMB_CARGA;
_001: NOP   0;
END_FUNCTION

FUNCTION "FC_Ctrl_Marcha" : VOID	// FC 10
VERSION : 0.1
VAR_TEMP
  FLG_COND_INICIAL : BOOL ;
  FLG_MENOR_MAX : BOOL ;
  FLG_MAYOR_MIN : BOOL ;
END_VAR
BEGIN
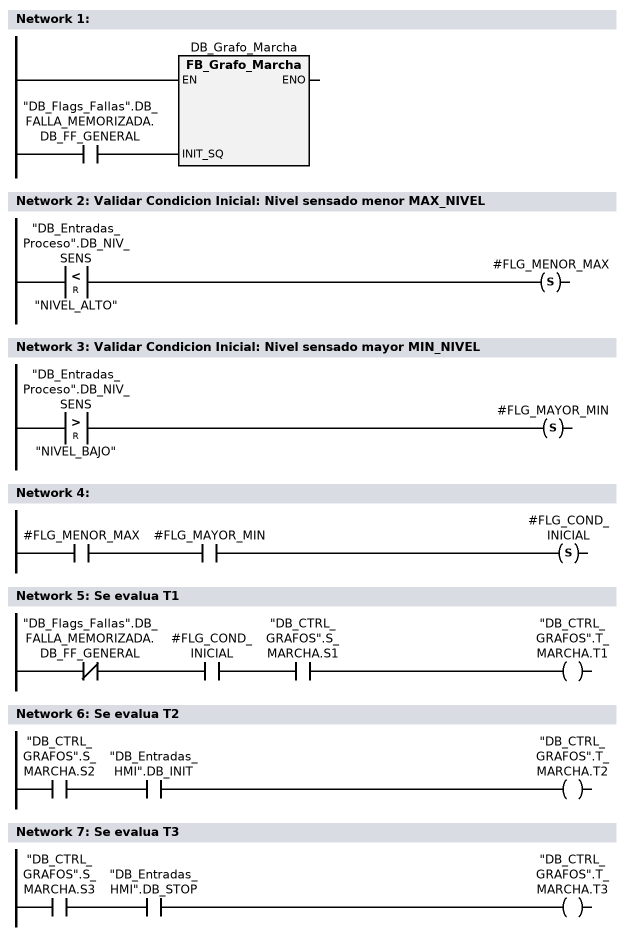
NETWORK
TITLE =
      A     "DB_Flags_Fallas".DB_FALLA_MEMORIZADA.DB_FF_GENERAL;
      =     L 1.1;
      BLD   103;
      CALL  "FB_Grafo_Marcha" , "DB_Grafo_Marcha" (
           INIT_SQ                  := L 1.1);
      NOP   0;
NETWORK
TITLE = Validar Condicion Inicial: Nivel sensado menor MAX_NIVEL
      L     "DB_Entradas_Proceso".DB_NIV_SENS;
      L     "NIVEL_ALTO";
      <R;
      S     #FLG_MENOR_MAX;
NETWORK
TITLE = Validar Condicion Inicial: Nivel sensado mayor MIN_NIVEL
      L     "DB_Entradas_Proceso".DB_NIV_SENS;
      L     "NIVEL_BAJO";
      >R;
      S     #FLG_MAYOR_MIN;
NETWORK
TITLE =
      A     #FLG_MENOR_MAX;
      A     #FLG_MAYOR_MIN;
      S     #FLG_COND_INICIAL;
NETWORK
TITLE = Se evalua T1
      AN    "DB_Flags_Fallas".DB_FALLA_MEMORIZADA.DB_FF_GENERAL;
      A     #FLG_COND_INICIAL;
      A     "DB_CTRL_GRAFOS".S_MARCHA.S1;
      =     "DB_CTRL_GRAFOS".T_MARCHA.T1;
NETWORK
TITLE = Se evalua T2
      A     "DB_CTRL_GRAFOS".S_MARCHA.S2;
      A     "DB_Entradas_HMI".DB_INIT;
      =     "DB_CTRL_GRAFOS".T_MARCHA.T2;
NETWORK
TITLE = Se evalua T3
      A     "DB_CTRL_GRAFOS".S_MARCHA.S3;
      A     "DB_Entradas_HMI".DB_STOP;
      =     "DB_CTRL_GRAFOS".T_MARCHA.T3;
END_FUNCTION

FUNCTION "FC_Ejecucion_PID" : VOID	// FC 11
VERSION : 0.1
VAR_INPUT
  SP_INT : REAL ;	//Set point
  PV_IN : REAL ;	//Es la variable a controlar (nivel sensado)
END_VAR
VAR_OUTPUT
  LMN : INT ;	//El valor manipulado, resultado del PID
END_VAR
VAR_TEMP
  TMP_REAL : REAL ;
  TMP_BCD : DINT ;
  TMP_LMN_P : REAL ;
  TMP_ERR : REAL ;
END_VAR
BEGIN
NETWORK
TITLE =
      A(;
      A     "FALSE";
      =     L 16.1;
      BLD   103;
      A     "FALSE";
      =     L 16.2;
      BLD   103;
      A     "TRUE";
      =     L 16.3;
      BLD   103;
      A     "TRUE";
      =     L 16.4;
      BLD   103;
      A     "FALSE";
      =     L 16.7;
      BLD   103;
      CALL  "CONT_C" , "DB_PID" (
           DIX 0.1                  := L 16.1,
           DIX 0.2                  := L 16.2,
           DIX 0.3                  := L 16.3,
           DIX 0.4                  := L 16.4,
           DIX 0.7                  := L 16.7,
           DID 2                    := L#100,
           DID 6                    := #SP_INT,
           DID 10                   := #PV_IN,
           DID 20                   := "DB_Entradas_HMI".DB_PID_KP,
           DID 24                   := "DB_Entradas_HMI".DB_PID_KI,
           DID 28                   := "DB_Entradas_HMI".DB_PID_KD,
           DID 56                   := L#1124744561,
           DID 60                   := L#0,
           DID 72                   := #TMP_REAL);
      A     BR;
      );
      JNB   _001;
      L     #TMP_REAL;
      T     #LMN;
_001: NOP   0;
END_FUNCTION

// FC 72: know-how protected block, not included

// FC 105: know-how protected block, not included

// FC 106: know-how protected block, not included

DATA_BLOCK "DB_Entradas_Proceso"	// DB 1
VERSION : 0.1
  STRUCT
   DB_NIV_SENS : REAL ;	//Entrada de nivel sensado (cuentas: 0 - 13824)
  END_STRUCT ;	
BEGIN
END_DATA_BLOCK

DATA_BLOCK "DB_Entradas_HMI"	// DB 2
VERSION : 0.1
  STRUCT
   DB_MOD_CTROL : INT ;	//2=PID ,1=ON/OFF y 0 = MANUAL
   DB_INIT : BOOL ;	//1 = Inicio del sistema
   DB_STOP : BOOL ;	//1 = Parada del sistema
   DB_SP_REF : REAL ;	//Setpoint de nivel de referencia
   DB_BANDA_HIST : REAL ;	//El valor de la banda de histeresis
   DB_CSG_BMB_PERT : INT ;	//Consigna de la bomba de perturbacion (vaciado). Valor del ciclo de 0 a 100.
   DB_CSG_BMB_CARGA : INT ;	//Consigna de la bomba de control (llenado). Valor del ciclo de 0 a 100.
   DB_MOD_PID : BOOL ;	//Flag que indica que el sistema opera en modo PID.
   DB_MOD_ONOFF : BOOL ;	//Flag que indica que el sistema opera en modo ON/OFF.
   DB_MOD_MANUAL : BOOL ;	//Flag que indica que el sistema opera en modo manual.
   PB_REC_FALLAS : BOOL ;	//Boton Pulsador de reconocimiento de fallas.
   DB_PID_KP : REAL ;	//La variable Kp del control PID. Proporcional
   DB_PID_KI : TIME ;	//La variable Ki del control PID. Integral
   DB_PID_KD : TIME ;	//La variable Kd del control PID. Derivativo
  END_STRUCT ;	
BEGIN
   DB_PID_KI := T#30S;
END_DATA_BLOCK

DATA_BLOCK "DB_Salidas_Proceso"	// DB 3
VERSION : 0.1
  STRUCT
   DB_BMB_CARGA : INT ;	//Señal de actuación sobre la bomba de carga del sistema (cuentas)
   DB_BMB_PERT : INT ;	//Señal de actuación sobre la bomba de perturbación del sistema (cuentas)
  END_STRUCT ;	
BEGIN
END_DATA_BLOCK

DATA_BLOCK "DB_Salidas_HMI"	// DB 4
VERSION : 0.1
  STRUCT
   DB_IND_ALARMA : BOOL ;	//Señal que indica que ocurrio una falla
   DB_COD_ALARMA : INT ;	//Codigo de la falla/s
   DB_NIVEL_MEDIDO : REAL ;	//Indicador del nivel del agua en el tanque
   DB_IND_MODO_MANUAL : BOOL ;	//Indicador de modo MANUAL.
   DB_IND_MODO_ON_OFF : BOOL ;	//Indicador de modo ON/OFF.
   DB_IND_MODO_PID : BOOL ;	//Indicador de modo PID.
  END_STRUCT ;	
BEGIN
END_DATA_BLOCK

DATA_BLOCK "DB_Flags_Fallas"	// DB 5
VERSION : 0.1
  STRUCT
   DB_FALLA_PRESENTE : STRUCT
    DB_FAR_SUP_NIV_MAX : BOOL ;	//Indicador de falla (Auto Reconocible): Se supero el nivel max.
    DB_FAR_SUP_NIV_MIN : BOOL ;	//Indicador de falla (Auto Reconocible): Por debajo del nivel minimo
    DB_FRO_BMB_CARGA : BOOL ;	//Indicador de falla (Reconocible por Ope.): Bomba de carga no funciona
    DB_FRO_SENSOR_NIV : BOOL ;	//Indicador de falla (Reconocible por Ope.): Sensor de nivel no funciona
    DB_FRO_SIN_CAUDAL_ENT : BOOL ;	//Indicador de falla (Reconocible por Ope.): Sin caudal de entrada
    DB_FF_GENERAL : BOOL ;	//Flag que indica que ocurrio alguna falla
   END_STRUCT ;
   DB_FALLA_MEMORIZADA : STRUCT
    DB_FAR_SUP_NIV_MAX : BOOL ;	//Indicador de falla: Se supero el nivel max.
    DB_FAR_SUP_NIV_MIN : BOOL ;	//Indicador de falla: Por debajo del nivel minimo
    DB_FRO_BMB_CARGA : BOOL ;	//Indicador de falla: Bomba de carga no funciona
    DB_FRO_SENSOR_NIV : BOOL ;	//Indicador de falla: Sensor de nivel no funciona
    DB_FRO_SIN_CAUDAL_ENT : BOOL ;	//Indicador de falla: Sin caudal de entrada
    DB_FF_GENERAL : BOOL ;	//Flag que indica que ocurrio alguna falla
   END_STRUCT ;
  END_STRUCT ;	
BEGIN
END_DATA_BLOCK

DATA_BLOCK "DB_Aux"	// DB 6
VERSION : 0.1
  STRUCT
   DB_CTAS_BMB_PERT : INT ;	//Valor en cuentas proporcional de la consigna del HMI
   DB_CTAS_BMB_CARGA : INT ;	//Valor en cuentas proporcional de la consigna del HMI
   DB_ERR_MOD_CTRL : BOOL ;	//Valor de modo de control incorrecto.
   DB_ERR_SP_REF : BOOL ;	//Valor de Set Point fuera de rango
   DB_ERR_BAND_HIST : BOOL ;	//Valor de banda de histeresis fuera de rango
   DB_ERR_CSG_BMB_CARGA : BOOL ;	//Valor de consigna bomba carga fuera de rango
   DB_ERR_CSG_BMB_PERT : BOOL ;	//Valor de consigna bomba perturbacion fuera de rango
   DB_FLG_BAND_HIST_SUP : BOOL ;	//Flag que indica que el nivel sensado supera la banda de histerisis
   DB_FLG_BAND_HIST_INF : BOOL ;	//Flag que indica que el nivel sensado esta por debajo de la banda de histerisis
  END_STRUCT ;	
BEGIN
END_DATA_BLOCK

DATA_BLOCK "DB_Grafo_Marcha"	// DB 7
VERSION : 0.0
"FB_Grafo_Marcha"
BEGIN
END_DATA_BLOCK

DATA_BLOCK "DB_Grafo_ON_OFF"	// DB 8
VERSION : 0.0
"FB_Grafo_ON_OFF"
BEGIN
END_DATA_BLOCK

DATA_BLOCK "DB_Grafo_PID"	// DB 9
VERSION : 0.0
"FB_Grafo_PID"
BEGIN
END_DATA_BLOCK

DATA_BLOCK "DB_CTRL_GRAFOS"	// DB 10
VERSION : 0.1
  STRUCT
   S_MARCHA : STRUCT
    S1 : BOOL ;	//Reposo
    S2 : BOOL ;	//OFF
    S3 : BOOL ;	//ON
    S4 : BOOL ;	//Ver si se usa !!!
   END_STRUCT ;
   T_MARCHA : STRUCT
    T1 : BOOL ;	//s1 a s2 (SALUD DEL SISTEMA)
    T2 : BOOL ;	//s2 a s3 (Init)
    T3 : BOOL ;	//s3 a s2 (Stop)
    T4 : BOOL ;	//Ver si se usa !!!
   END_STRUCT ;
   S_ONOFF : STRUCT
    S1 : BOOL ;	//Reposo
    S2 : BOOL ;	//Bomba Detenida
    S3 : BOOL ;	//Bomba Funcionando
    S4 : BOOL ;	//Ver si se usa !!!
   END_STRUCT ;
   T_ONOFF : STRUCT
    T1 : BOOL ;	//s1 a s2 (ON y Modo = ONOFF)
    T2 : BOOL ;	//s2 a s3 (Nivel < Banda Hist. Inferior)
    T3 : BOOL ;	//s3 a s2 (Nivel > Banda Hist. Superior)
    T4 : BOOL ;	//Ver si se usa !!!
   END_STRUCT ;
   S_PID : STRUCT
    S1 : BOOL ;	//Reposo
    S2 : BOOL ;	//Modo Manual
    S3 : BOOL ;	//Modo PID
    S4 : BOOL ;	//Ver si se usa !!!
   END_STRUCT ;
   T_PID : STRUCT
    T1 : BOOL ;	//s1 a s2 (ON y Modo = Manual)
    T2 : BOOL ;	//s2 a s3 (Nivel < Banda Hist. Inferior)
    T3 : BOOL ;	//s3 a s2 (Nivel > Banda Hist. Superior)
    T4 : BOOL ;	//Ver si se usa !!!
   END_STRUCT ;
  END_STRUCT ;	
BEGIN
END_DATA_BLOCK

DATA_BLOCK "DB_PID"	// DB 11
AUTHOR : SIMATIC
FAMILY : ICONT
VERSION : 0.1
"CONT_C"
BEGIN
END_DATA_BLOCK

ORGANIZATION_BLOCK "Programa Principal"	// OB 1
TITLE = "Main Program Sweep (Cycle)"
VERSION : 0.1
VAR_TEMP
  OB1_EV_CLASS : BYTE ;	//Bits 0-3 = 1 (Coming event), Bits 4-7 = 1 (Event class 1)
  OB1_SCAN_1 : BYTE ;	//1 (Cold restart scan 1 of OB 1), 3 (Scan 2-n of OB 1)
  OB1_PRIORITY : BYTE ;	//Priority of OB Execution
  OB1_OB_NUMBR : BYTE ;	//1 (Organization block 1, OB1)
  OB1_RESERVED_1 : BYTE ;	//Reserved for system
  OB1_RESERVED_2 : BYTE ;	//Reserved for system
  OB1_PREV_CYCLE : INT ;	//Cycle time of previous OB1 scan (milliseconds)
  OB1_MIN_CYCLE : INT ;	//Minimum cycle time of OB1 (milliseconds)
  OB1_MAX_CYCLE : INT ;	//Maximum cycle time of OB1 (milliseconds)
  OB1_DATE_TIME : DATE_AND_TIME ;	//Date and time OB1 started
END_VAR
BEGIN
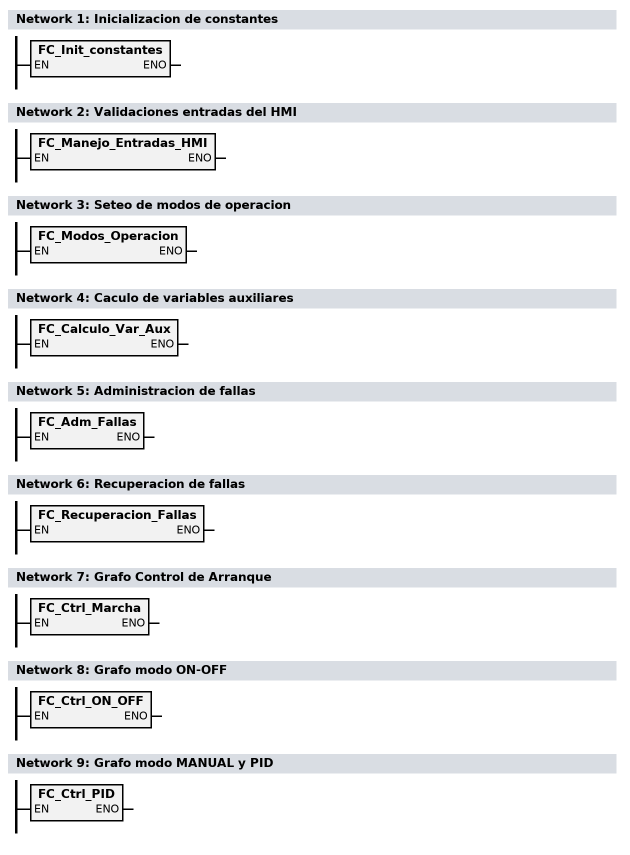
NETWORK
TITLE = Inicializacion de constantes
      CALL  "FC_Init_constantes";
      NOP   0;
NETWORK
TITLE = Validaciones entradas del HMI
      CALL  "FC_Manejo_Entradas_HMI";
      NOP   0;
NETWORK
TITLE = Seteo de modos de operacion
      CALL  "FC_Modos_Operacion";
      NOP   0;
NETWORK
TITLE = Caculo de variables auxiliares
      CALL  "FC_Calculo_Var_Aux";
      NOP   0;
NETWORK
TITLE = Administracion de fallas
      CALL  "FC_Adm_Fallas";
      NOP   0;
NETWORK
TITLE = Recuperacion de fallas
      CALL  "FC_Recuperacion_Fallas";
      NOP   0;
NETWORK
TITLE = Grafo Control de Arranque
      CALL  "FC_Ctrl_Marcha";
      NOP   0;
NETWORK
TITLE = Grafo modo ON-OFF
      CALL  "FC_Ctrl_ON_OFF";
      NOP   0;
NETWORK
TITLE = Grafo modo MANUAL y PID
      CALL  "FC_Ctrl_PID";
      NOP   0;
END_ORGANIZATION_BLOCK

ORGANIZATION_BLOCK "CYC_INT5"	// OB 35
TITLE = "Cyclic Interrupt"
VERSION : 0.1
VAR_TEMP
  OB35_EV_CLASS : BYTE ;	//Bits 0-3 = 1 (Coming event), Bits 4-7 = 1 (Event class 1)
  OB35_STRT_INF : BYTE ;	//16#36 (OB 35 has started)
  OB35_PRIORITY : BYTE ;	//Priority of OB Execution
  OB35_OB_NUMBR : BYTE ;	//35 (Organization block 35, OB35)
  OB35_RESERVED_1 : BYTE ;	//Reserved for system
  OB35_RESERVED_2 : BYTE ;	//Reserved for system
  OB35_PHASE_OFFSET : WORD ;	//Phase offset (msec)
  OB35_RESERVED_3 : INT ;	//Reserved for system
  OB35_EXC_FREQ : INT ;	//Frequency of execution (msec)
  OB35_DATE_TIME : DATE_AND_TIME ;	//Date and time OB35 started
  RV : WORD ;
END_VAR
BEGIN
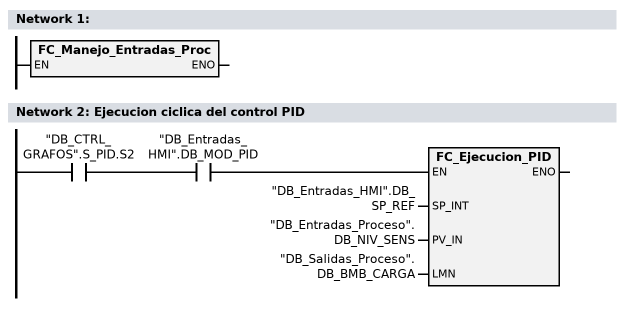
NETWORK
TITLE =
      CALL  "FC_Manejo_Entradas_Proc";
      NOP   0;
NETWORK
TITLE = Ejecucion ciclica del control PID
      A     "DB_CTRL_GRAFOS".S_PID.S2;
      A     "DB_Entradas_HMI".DB_MOD_PID;
      JNB   _001;
      CALL  "FC_Ejecucion_PID" (
           SP_INT                   := "DB_Entradas_HMI".DB_SP_REF,
           PV_IN                    := "DB_Entradas_Proceso".DB_NIV_SENS,
           LMN                      := "DB_Salidas_Proceso".DB_BMB_CARGA);
_001: NOP   0;
END_ORGANIZATION_BLOCK

SYMBOL_TABLE
"DB_Entradas_Proceso"	DB 1	DB 1
"DB_Entradas_HMI"	DB 2	DB 2
"DB_Salidas_Proceso"	DB 3	DB 3
"DB_Salidas_HMI"	DB 4	DB 4
"DB_Flags_Fallas"	DB 5	DB 5
"DB_Aux"	DB 6	DB 6	// DB de variables auxiliares
"DB_Grafo_Marcha"	DB 7	FB 1
"DB_Grafo_ON_OFF"	DB 8	FB 2
"DB_Grafo_PID"	DB 9	FB 3
"DB_CTRL_GRAFOS"	DB 10	DB 10	// DB Global de estados y transiciones de grafos
"DB_PID"	DB 11	FB 41
"DB_Parametrizaion_PID"	DB 12	DB 12
"FB_Grafo_Marcha"	FB 1	FB 1
"FB_Grafo_ON_OFF"	FB 2	FB 2
"FB_Grafo_PID"	FB 3	FB 3
"CONT_C"	FB 41	FB 41	// Continuous Control
"FC_Init_constantes"	FC 1	FC 1
"FC_Manejo_Entradas_Proc"	FC 2	FC 2
"FC_Manejo_Entradas_HMI"	FC 3	FC 3
"FC_Modos_Operacion"	FC 4	FC 4
"FC_Calculo_Var_Aux"	FC 5	FC 5	// Funcion que calcula variables aux.
"FC_Adm_Fallas"	FC 6	FC 6	// Funcion que verifica fallas del sistema
"FC_Recuperacion_Fallas"	FC 7	FC 7	// Recuperacion automatica de fallas
"FC_Ctrl_ON_OFF"	FC 8	FC 8
"FC_Ctrl_PID"	FC 9	FC 9
"FC_Ctrl_Marcha"	FC 10	FC 10
"FC_Ejecucion_PID"	FC 11	FC 11
"FC_Manejo_Salidas_HMI"	FC 12	FC 12
"FC_Manejo_Salida_Proceso"	FC 13	FC 13
"G7_STD_3"	FC 72	FC 72
"Stack (LIFO)"	FC 93	FC 93	// Stack (last in first out)
"SCALE"	FC 105	FC 105	// Scaling Values
"UNSCALE"	FC 106	FC 106	// Unscaling Values
"FALLA_BMB"	I 4.0	BOOL	// Señal (simulada) de falla de bomba
"NIV_SENS"	IW 108	INT	// Nivel sensado del liquido en el tacho (Cuentas)
"FALSE"	M 0.0	BOOL
"TRUE"	M 0.1	BOOL
"ALTURA_TACHO"	MD 1	REAL	// Altura del tacho (cm)
"NIVEL_ALTO"	MD 3	REAL	// Nivel maximo de agua en el tacho
"NIVEL_BAJO"	MD 5	REAL	// Minimo nivel de agua en el tacho
"Programa Principal"	OB 1	OB 1
"CYC_INT5"	OB 35	OB 35	// Cyclic Interrupt 5
"SALIDA_HL"	Q 4.0	BOOL	// Indicacion de nivel alto (HL)
"SALIDA_LL"	Q 4.1	BOOL	// Indicación de nivel bajo (LL)
"LUZ_MODO_OPER"	Q 4.2	BOOL	// Indicacion del modo de operacion (MANUAL-ON/OFF-PID)
"BMB_CARGA"	QW 100	INT	// Señal de actuación sobre la bomba de carga del sistema. Rango entre 0 y 5 V.
"BMB_PERT"	QW 102	INT	// Señal de actuación sobre la bomba de perturbación (vaciado) del sistema.
"ALARM_SQ"	SFC 17	SFC 17	// Generate Block-Related Messages with Acknowledgment
"ALARM_S"	SFC 18	SFC 18	// Generate Permanently Acknowledged Block-Related Messages
"WR_USMSG"	SFC 52	SFC 52	// Write a User-Defined Diagnostic Event to the Diagnostic Buffer
"TIME_TCK"	SFC 64	SFC 64	// Read the System Time
"VAT_SIM"	VAT 1	
END_SYMBOL_TABLE
